(* IEC 61131-3 sources: Word/plc-course/18-hmi-and-scada/labs/solutions, 2 files *)

(* ---- 18-1-command-handshake.st ---- *)
(* Lab 18-1: HMI command handshake for transfer pump P-101.
   Module 18 (HMI and SCADA). REFERENCE SOLUTION - try the lab yourself first.

   The HMI talks to the PLC over Modbus TCP. It never switches the pump
   directly: it writes a COMMAND WORD (one bit per command), and the PLC
   decides. The PLC acts on each command exactly once, clears the word
   ("PLC clears the command"), reports its state in a STATUS WORD, and
   explains every refusal with a REJECT CODE.

   In the OpenPLC Runtime v3, %MW0..%MW1023 are Modbus holding registers
   1024..2047, so an HMI would find HmiCmd at holding register 1024. Newer
   OpenPLC releases let you size the register blocks, so check the Modbus
   address table that your version shows. *)

PROGRAM CmdHandshake
  VAR (* field I/O *)
    OverloadOK_NC AT %IX0.0 : BOOL;  (* Overload relay contact, NC: TRUE = healthy *)
    SuctionOK     AT %IX0.1 : BOOL;  (* Start permissive: feed-tank level above low (LSL-101) *)
    PumpRun       AT %QX0.0 : BOOL;  (* Pump contactor *)
  END_VAR
  VAR (* HMI interface - memory words the HMI reads and writes *)
    HmiCmd     AT %MW0 : WORD;       (* HMI -> PLC: command bits. HMI sets, PLC clears *)
    HmiSts     AT %MW1 : WORD;       (* PLC -> HMI: status bits *)
    RejectCode AT %MW2 : INT;        (* PLC -> HMI: result of the last command, 0 = accepted *)
    SpeedReq   AT %MW3 : INT;        (* HMI -> PLC: requested speed, % *)
    SpeedSP    AT %MW4 : INT := 50;  (* PLC -> HMI: active speed setpoint, % *)
  END_VAR
  VAR CONSTANT
    (* Command bits in HmiCmd *)
    CMD_START   : WORD := 16#0001;
    CMD_STOP    : WORD := 16#0002;
    CMD_RESET   : WORD := 16#0004;
    CMD_APPLY   : WORD := 16#0008;
    CMD_DEFINED : WORD := 16#000F;   (* every bit that means something *)
    (* Status bits in HmiSts *)
    STS_RUNNING  : WORD := 16#0001;
    STS_FAULTED  : WORD := 16#0002;
    STS_READY    : WORD := 16#0004;
    STS_PERMOK   : WORD := 16#0008;
    STS_REJECTED : WORD := 16#0010;
    (* Reject codes *)
    REJ_NONE       : INT := 0;
    REJ_UNKNOWN    : INT := 1;
    REJ_FAULTED    : INT := 2;
    REJ_NO_PERMIT  : INT := 3;
    REJ_FAULT_HERE : INT := 4;
    REJ_SP_RANGE   : INT := 5;
    (* Engineered speed limits, % *)
    SPEED_MIN : INT := 30;
    SPEED_MAX : INT := 100;
  END_VAR
  VAR
    FirstScanDone : BOOL;            (* FALSE only on the first scan after power-up *)
    Cmd           : WORD;            (* this scan's snapshot of HmiCmd *)
    Result        : INT;             (* reject code for this command word *)
    LastReject    : INT;             (* result of the last command word, kept *)
    Faulted       : BOOL;            (* latched overload fault *)
    Running       : BOOL;            (* run latch *)
    Sts           : WORD;            (* status word being built *)
    ActiveSpeed   : INT := 50;       (* the setpoint in use. SpeedSP is only a copy for
                                        the HMI, so a stray write to it changes nothing *)
  END_VAR

  (* 1. Take a snapshot of the command word and clear it at once.
        Everything below works on the snapshot, so the command is acted on
        exactly once, and a comms drop can never leave a bit "stuck on". *)
  Cmd := HmiCmd;
  HmiCmd := 16#0000;

  (* A command that is already waiting on the first scan was written
     before the power cut (or is left in retentive memory). Executing it now
     could start the pump unexpectedly, so it is discarded. *)
  IF NOT FirstScanDone THEN
    Cmd := 16#0000;
    FirstScanDone := TRUE;
  END_IF;

  (* 2. Protection first: the overload latches a fault at any time. *)
  IF NOT OverloadOK_NC THEN
    Faulted := TRUE;
  END_IF;

  (* 3. Handle the command word (only when there is one). *)
  IF Cmd <> 16#0000 THEN
    Result := REJ_NONE;

    IF (Cmd AND CMD_STOP) <> 16#0000 THEN
      (* Stop wins over everything and is never refused. *)
      Running := FALSE;

    ELSIF (Cmd AND NOT CMD_DEFINED) <> 16#0000 THEN
      (* A bit we do not understand: do nothing rather than guess. *)
      Result := REJ_UNKNOWN;

    ELSE
      (* Reset first, so that Reset + Start in one word works. *)
      IF (Cmd AND CMD_RESET) <> 16#0000 THEN
        IF OverloadOK_NC THEN
          Faulted := FALSE;          (* reset never starts the pump *)
        ELSIF Result = REJ_NONE THEN
          Result := REJ_FAULT_HERE;
        END_IF;
      END_IF;

      IF (Cmd AND CMD_START) <> 16#0000 THEN
        IF Faulted THEN
          IF Result = REJ_NONE THEN Result := REJ_FAULTED; END_IF;
        ELSIF NOT SuctionOK THEN
          IF Result = REJ_NONE THEN Result := REJ_NO_PERMIT; END_IF;
        ELSE
          Running := TRUE;           (* already running: accepted, no change *)
        END_IF;
      END_IF;

      IF (Cmd AND CMD_APPLY) <> 16#0000 THEN
        (* Written as "inside the range" so that anything odd is refused. *)
        IF SpeedReq >= SPEED_MIN AND SpeedReq <= SPEED_MAX THEN
          ActiveSpeed := SpeedReq;
        ELSIF Result = REJ_NONE THEN
          Result := REJ_SP_RANGE;    (* the old setpoint stays in use *)
        END_IF;
      END_IF;
    END_IF;

    LastReject := Result;            (* kept until the next command word *)
  END_IF;

  (* 4. Interlocks: a trip or a lost permissive stops the pump. It does not
        restart when the condition clears - that needs a new Start. *)
  IF Faulted OR NOT SuctionOK THEN
    Running := FALSE;
  END_IF;
  PumpRun := Running;

  (* 5. Publish the status for the HMI. These registers are written every
        scan, so nothing written into them from outside can stick. *)
  SpeedSP := ActiveSpeed;
  RejectCode := LastReject;
  Sts := 16#0000;
  IF Running THEN Sts := Sts OR STS_RUNNING; END_IF;
  IF Faulted THEN Sts := Sts OR STS_FAULTED; END_IF;
  IF NOT Running AND NOT Faulted AND SuctionOK THEN Sts := Sts OR STS_READY; END_IF;
  IF SuctionOK THEN Sts := Sts OR STS_PERMOK; END_IF;
  IF LastReject <> REJ_NONE THEN Sts := Sts OR STS_REJECTED; END_IF;
  HmiSts := Sts;
END_PROGRAM

CONFIGURATION Config0
  RESOURCE Res0 ON PLC
    TASK MainTask(INTERVAL := T#10ms, PRIORITY := 0);
    PROGRAM Inst0 WITH MainTask : CmdHandshake;
  END_RESOURCE
END_CONFIGURATION

(* ---- 18-2-mode-manager.st ---- *)
(* Lab 18-2: Mode manager for wet-well pump P-201.
   Module 18 (HMI and SCADA). REFERENCE SOLUTION - try the lab yourself first.

   Modes:   Off / Manual / Auto, chosen from the HMI (Remote) only.
   Source:  Local (field control station LCS-201) or Remote (HMI/SCADA),
            chosen by the key selector at the pump.
   The mode manager decides who may command the pump, refuses requests that
   are not allowed (with a reason code), and makes every mode and source
   change bumpless: the pump only changes state when the NEW owner wants it.

   Training exercise only. On a real plant, dry-run protection and the local
   stop are usually hardwired as well as handled in the PLC. *)

PROGRAM ModeManager
  VAR (* field I/O *)
    LocalSel       AT %IX0.0 : BOOL;  (* Local/Remote selector at LCS-201: TRUE = Local *)
    LocalStartPB   AT %IX0.1 : BOOL;  (* Local Start push-button, NO *)
    LocalStopPB_NC AT %IX0.2 : BOOL;  (* Local Stop push-button, NC: TRUE while not pressed *)
    RunPermit      AT %IX0.3 : BOOL;  (* LSLL-201: TRUE while level is above low-low *)
    MotorRun       AT %QX0.0 : BOOL;  (* Pump contactor *)
  END_VAR
  VAR (* HMI interface - memory words the HMI reads and writes *)
    ModeReq    AT %MW0 : INT;         (* HMI -> PLC: 0 none, 1 Off, 2 Manual, 3 Auto. PLC clears *)
    MotorCmd   AT %MW1 : INT;         (* HMI -> PLC: 0 none, 1 Start, 2 Stop. PLC clears *)
    ActiveMode AT %MW2 : INT := 1;    (* PLC -> HMI: 1 Off, 2 Manual, 3 Auto *)
    RejectCode AT %MW3 : INT;         (* PLC -> HMI: result of the last HMI request *)
  END_VAR
  VAR (* from the level controller (other code; set by the test in this lab) *)
    AutoDemand    : BOOL;             (* TRUE = the level controller wants the pump *)
    AutoAvailable : BOOL;             (* TRUE = LT-201 healthy, so Auto can work *)
  END_VAR
  VAR CONSTANT
    MODE_OFF  : INT := 1;
    MODE_MAN  : INT := 2;
    MODE_AUTO : INT := 3;
    CMD_START : INT := 1;
    CMD_STOP  : INT := 2;
    REJ_NONE       : INT := 0;
    REJ_LOCAL      : INT := 1;        (* Local selected: the HMI has no control *)
    REJ_INVALID    : INT := 2;        (* value not defined *)
    REJ_NO_AUTO    : INT := 3;        (* Auto not possible now *)
    REJ_NOT_MANUAL : INT := 4;        (* Start is only allowed in Manual *)
    REJ_NO_PERMIT  : INT := 5;        (* start permissive missing *)
  END_VAR
  VAR
    FirstScanDone : BOOL;             (* FALSE only on the first scan after power-up *)
    Req        : INT;                 (* snapshot of ModeReq *)
    Cmd        : INT;                 (* snapshot of MotorCmd *)
    Result     : INT;                 (* first refusal this scan, or 0 *)
    LastReject : INT;                 (* result of the last HMI request, kept *)
    IsLocal    : BOOL;
    StopHeld   : BOOL;                (* local Stop pressed (or its wire broken) *)
    CanRun     : BOOL;                (* all run permissives healthy *)
    Running    : BOOL;                (* the run state; in Auto it tracks AutoDemand *)
    Mode       : INT := 1;            (* the real mode. ActiveMode is only a copy for
                                         the HMI, so a stray write to it changes nothing *)
  END_VAR

  (* 1. Snapshot the HMI requests and clear them: each is handled once. *)
  Req := ModeReq;
  ModeReq := 0;
  Cmd := MotorCmd;
  MotorCmd := 0;

  (* A request already waiting on the first scan was written before a power
     cut or a download. Acting on it now could put the pump in Auto and
     start it with nobody watching, so it is discarded (as in Lab 18-1). *)
  IF NOT FirstScanDone THEN
    Req := 0;
    Cmd := 0;
    FirstScanDone := TRUE;
  END_IF;

  IsLocal := LocalSel;
  StopHeld := NOT LocalStopPB_NC;
  CanRun := RunPermit AND NOT StopHeld;

  (* 2. Control source. Local always means local manual control. The run
        state is not touched, so the transfer is bumpless both ways. *)
  IF IsLocal THEN
    Mode := MODE_MAN;
  END_IF;

  (* 3. HMI requests. The mode request is handled before the motor command,
        and RejectCode reports the first refusal. *)
  IF Req <> 0 OR Cmd <> 0 THEN
    Result := REJ_NONE;

    IF Req <> 0 THEN
      IF IsLocal THEN
        Result := REJ_LOCAL;
      ELSIF Req = MODE_OFF OR Req = MODE_MAN THEN
        Mode := Req;                  (* Manual keeps the pump as it is *)
      ELSIF Req = MODE_AUTO THEN
        IF AutoAvailable AND NOT StopHeld THEN
          Mode := MODE_AUTO;          (* the pump now follows AutoDemand *)
        ELSE
          Result := REJ_NO_AUTO;
        END_IF;
      ELSE
        Result := REJ_INVALID;
      END_IF;
    END_IF;

    IF Cmd = CMD_STOP THEN
      (* A stop is obeyed from any source and in any mode. In Auto it also
         hands the pump to Manual, so the demand cannot restart it. *)
      Running := FALSE;
      IF Mode = MODE_AUTO THEN
        Mode := MODE_MAN;
      END_IF;
    ELSIF Cmd <> 0 THEN
      IF IsLocal THEN
        IF Result = REJ_NONE THEN Result := REJ_LOCAL; END_IF;
      ELSIF Cmd <> CMD_START THEN
        IF Result = REJ_NONE THEN Result := REJ_INVALID; END_IF;
      ELSIF Mode <> MODE_MAN THEN
        IF Result = REJ_NONE THEN Result := REJ_NOT_MANUAL; END_IF;
      ELSIF NOT CanRun THEN
        IF Result = REJ_NONE THEN Result := REJ_NO_PERMIT; END_IF;
      ELSE
        Running := TRUE;
      END_IF;
    END_IF;

    LastReject := Result;             (* kept until the next request *)
  END_IF;

  (* 4. Local push-buttons. Start works only in Local; Stop is covered by
        CanRun below and works everywhere. *)
  IF IsLocal AND LocalStartPB AND CanRun THEN
    Running := TRUE;
  END_IF;

  (* 5. Auto drops to Manual when it can no longer work (mode shedding, the
        pump keeps its state) or when someone presses the local Stop. *)
  IF Mode = MODE_AUTO AND (NOT AutoAvailable OR StopHeld) THEN
    Mode := MODE_MAN;
  END_IF;

  (* 6. The run state for each mode. In Auto, Running is overwritten with the
        demand every scan, so it always holds the pump's real state; that is
        what makes Auto -> Manual bumpless. *)
  IF Mode = MODE_OFF THEN
    Running := FALSE;
  ELSIF Mode = MODE_AUTO THEN
    Running := AutoDemand;
  END_IF;

  (* 7. Permissives win in every mode. In Manual the pump stays off when the
        permissive returns; in Auto it follows the demand again. *)
  IF NOT CanRun THEN
    Running := FALSE;
  END_IF;
  MotorRun := Running;

  (* 8. Publish the status for the HMI. These registers are written every
        scan, so nothing written into them from outside can stick. *)
  ActiveMode := Mode;
  RejectCode := LastReject;
END_PROGRAM

CONFIGURATION Config0
  RESOURCE Res0 ON PLC
    TASK MainTask(INTERVAL := T#10ms, PRIORITY := 0);
    PROGRAM Inst0 WITH MainTask : ModeManager;
  END_RESOURCE
END_CONFIGURATION
